(* IEC 61131-3 sources: Warcbot/Robot-programy, 4 files *)

(* ---- gohome.st ---- *)
VAR {AT 'MotionCtrl'}
    Done {ACCESS 'STMotionDone'}: BOOL;
END_VAR

VAR
    Home : McAxisTargetType := (JointAxis:=[0,0,-90,0,90,0]);
END_VAR

PROGRAM _MAIN
    Done := FALSE;
    Feedrate(500);

    MoveA(Home);
    WaitEndMove();
    Done := TRUE;
END_PROGRAM

(* ---- move.st ---- *)
VAR {AT 'MotionCtrl'}
    StartPoint {ACCESS 'STMotionStartPoint'}: McPointType;
    EndPoint {ACCESS 'STMotionEndPoint'}: McPointType;
    HomePoint {ACCESS 'STMotionHomePoint'}: McPointType;
    Done {ACCESS 'STMotionDone'}: BOOL;
END_VAR

VAR {AT PLC}
    doMagnet : BOOL;
END_VAR

VAR
    Offs : McPosType := (Z:=20);

    StartPointOffs : McPointType;
    EndPointOffs : McPointType;
END_VAR

PROGRAM _MAIN
    Done := FALSE;
    Feedrate(5000);

    StartPointOffs := StartPoint;
    StartPointOffs.Pos.Z := StartPointOffs.Pos.Z + Offs.Z;
    EndPointOffs := EndPoint;
    EndPointOffs.Pos.Z := EndPointOffs.Pos.Z + Offs.Z;

    MoveJ(StartPointOffs);
    Feedrate(500);
    MoveL(StartPoint);
    Feedrate(5000);
    WaitEndMove();
    doMagnet := TRUE;
    //WaitUntil(MagnetStatus);
    MoveL(StartPointOffs); // zapytac sie czy tutaj da sie dac StartPoint + Offs, dla krotszego kodu

    //MoveJ(HomePoint);

    MoveJ(EndPointOffs);
    Feedrate(500);
    MoveL(EndPoint);
    Feedrate(5000);
    WaitEndMove();
    doMagnet := FALSE;
    //WaitUntil(NOT MagnetStatus);
    MoveL(EndPointOffs);

    MoveJ(HomePoint);

    WaitEndMove();
    Done := TRUE;
END_PROGRAM

(* ---- moveAB.st ---- *)
VAR {AT 'MotionCtrl'}
    StartPoint {ACCESS 'STMotionStartPoint'}: McPointType;
    EndPoint {ACCESS 'STMotionEndPoint'}: McPointType;
    Done {ACCESS 'STMotionDone'}: BOOL;

    HighFeedrate {ACCESS 'STMotionHighFeedrate'}: LREAL;
    LowFeedrate {ACCESS 'STMotionLowFeedrate'}: LREAL;
END_VAR

VAR {AT PLC}
    doMagnet : BOOL;
    UserFrame {ACCESS 'gUserFrame'}: McFrameType;
END_VAR

VAR
    Offs : McPosType := (Z:=20);

    StartPointOffs : McPointType;
    EndPointOffs : McPointType;
END_VAR

PROGRAM _MAIN
    Done := FALSE;
    //SetPCS(OH::gUserFrame);
    Feedrate(HighFeedrate);

    StartPointOffs := StartPoint;
    StartPointOffs.Pos.Z := StartPointOffs.Pos.Z + Offs.Z;
    EndPointOffs := EndPoint;
    EndPointOffs.Pos.Z := EndPointOffs.Pos.Z + Offs.Z;

    MoveJ(StartPointOffs);
    Feedrate(LowFeedrate);
    MoveL(StartPoint);
    WaitEndMove();
    doMagnet := TRUE;
    WaitTime(1);
    MoveL(StartPointOffs); // zapytac sie czy tutaj da sie dac StartPoint + Offs, dla krotszego kodu
    Feedrate(HighFeedrate);

    //MoveJ(HomePoint);

    MoveJ(EndPointOffs);
    Feedrate(LowFeedrate);
    MoveL(EndPoint);
    WaitEndMove();
    doMagnet := FALSE;
    WaitTime(1);
    MoveL(EndPointOffs);
    Feedrate(HighFeedrate);

    WaitEndMove();
    Done := TRUE;
END_PROGRAM

(* ---- test.st ---- *)
VAR
    Point_10 : McPointType :=
END_VAR

MoveL()
